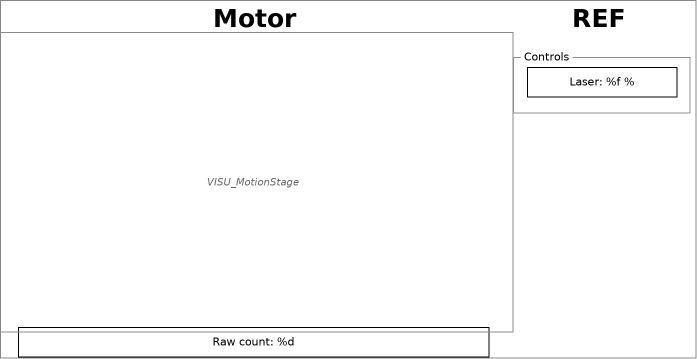
VISUALIZATION Visualization  // 697x359
    Label (14,3 482x30), "Motor"
    Label (503,3 192x30), "REF"
    Rectangle (18,327 471x30), "Raw count: %d", text variable: Main.iAdjustedEncoder
    GroupBox (513,49 177x64), "Controls"
        Rectangle (14,18 150x30), "Laser: %f %", text variable: Main.fbREF.fbLaser.fLaserPercent
            OnMouseDown: write the text variable via Default, min 0, max 100
    Frame (-7,32 520x300)
        shows VISU_MotionStage(VisuMotionStage := Main.M1, Extras := Main.M1_Extras)
END_VISUALIZATION

(* stored: Version 1.1.0.1, ProductVersion 3.1.4022.12
   Visu Visualization: Id {af2f16f4-e7e7-4019-a84a-cc323e4115d2} *)
